// TIA Portal V16 export
// export: Created 2023-01-04T15:44:08.5124159Z, ExportSetting WithDefaults, DisplayName Totally Integrated Automation Portal, DisplayVersion V16, DisplayName TIA Portal Version Control Interface, DisplayVersion V16, DisplayName TIA Portal Openness, DisplayVersion V16, DisplayName STEP 7 Professional, DisplayVersion V16, DisplayName STEP 7 Safety, DisplayVersion V16, DisplayName WinCC Advanced, DisplayVersion V16
FUNCTION "Scalling_Output" : Void   // FC2, FBD
{ S7_Optimized_Access := 'TRUE' }
VERSION : 0.1
// stored: AutoNumber true, IsIECCheckEnabled false, SetENOAutomatically false, UDAEnableTagReadback false
   VAR_INPUT
      IN_Min : Int;
      Input : Int;
      IN_Max : Int;
      Out_Min : Int;
      Out_Max : Int;
   END_VAR
   VAR_OUTPUT
      Output : Int;
   END_VAR
   VAR_TEMP
      Normed : Real;
   END_VAR
BEGIN

REGION Network 1
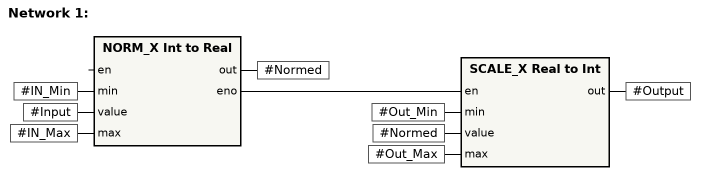
   #Normed := NORM_X(MIN := #IN_Min, VALUE := #Input, MAX := #IN_Max);
   #Output := SCALE_X(MIN := #Out_Min, VALUE := #Normed, MAX := #Out_Max);
END_REGION
END_FUNCTION
